VAR_GLOBAL

{attribute 'TcLinkTo' := 		'.q_xPress_OK		:= 	TIPC^txi_sxr_vac^txi_sxr_vac Instance^FSV_task Inputs^GVL_TXI_VAC_VFS.TV2K3_VFS_01.i_xPress_OK;
                                 .q_xOPN_SW			:=  TIPC^txi_sxr_vac^txi_sxr_vac Instance^FSV_task Inputs^GVL_TXI_VAC_VFS.TV2K3_VFS_01.i_xOPN_SW;
                                 .q_xCLS_SW			:=  TIPC^txi_sxr_vac^txi_sxr_vac Instance^FSV_task Inputs^GVL_TXI_VAC_VFS.TV2K3_VFS_01.i_xCLS_SW;
                                 .q_xVAC_FAULT_Reset:= 	TIPC^txi_sxr_vac^txi_sxr_vac Instance^FSV_task Inputs^GVL_TXI_VAC_VFS.TV2K3_VFS_01.i_xVAC_FAULT_Reset;
                                 .q_xOverrideMode	:= 	TIPC^txi_sxr_vac^txi_sxr_vac Instance^FSV_task Inputs^GVL_TXI_VAC_VFS.TV2K3_VFS_01.i_xOverrideMode;
                                 .q_xOverrideOpen	:= 	TIPC^txi_sxr_vac^txi_sxr_vac Instance^FSV_task Inputs^GVL_TXI_VAC_VFS.TV2K3_VFS_01.i_xOverrideOpen;
                                 .i_xTrigger		:=	TIPC^txi_sxr_vac^txi_sxr_vac Instance^FSV_task Outputs^GVL_TXI_VAC_VFS.TV2K3_VFS_01.q_xTrigger;
                                 .i_xVFS_Open		:=	TIPC^txi_sxr_vac^txi_sxr_vac Instance^FSV_task Outputs^GVL_TXI_VAC_VFS.TV2K3_VFS_01.q_xVFS_Open;
                                 .i_xVFS_Closed		:=	TIPC^txi_sxr_vac^txi_sxr_vac Instance^FSV_task Outputs^GVL_TXI_VAC_VFS.TV2K3_VFS_01.q_xVFS_Closed;
                                 .i_xVAC_FAULT_OK	:=  TIPC^txi_sxr_vac^txi_sxr_vac Instance^FSV_task Outputs^GVL_TXI_VAC_VFS.TV2K3_VFS_01.q_xVAC_FAULT_OK;
                                 .i_xMPS_OK			:=  TIPC^txi_sxr_vac^txi_sxr_vac Instance^FSV_task Outputs^GVL_TXI_VAC_VFS.TV2K3_VFS_01.q_xMPS_OK;
                                 .i_eVFS_State		:=	TIPC^txi_sxr_vac^txi_sxr_vac Instance^FSV_task Outputs^GVL_TXI_VAC_VFS.TV2K3_VFS_01.q_eVFS_State;
'}
TV2K3_VFS_01_Interface : FB_VFS_Interface;

{attribute 'pytmc' := 'pv: TV2K3:VFS:01'}
{attribute 'TcLinkTo' := 	'
        .q_xClose_A	:=	TIIB[H1K3S01-DRL-01 E1 (EL2202)]^Channel 1^Output;
        .q_xClose_B	:=	TIIB[H1K3S01-DRL-01 E1 (EL2202)]^Channel 2^Output;
        .q_xClose_C	:=	TIIB[H1K3S01-DRL-01 E2 (EL2202)]^Channel 1^Output;
        .q_xOPN_DO	:=	TIIB[H1K3S01-DRL-01 E2 (EL2202)]^Channel 2^Output;
        .i_xClsLS	:=	TIIB[H1K3S01-DRL-01 E3 (EL1004)]^Channel 1^Input;
        .i_xOpnLS	:=	TIIB[H1K3S01-DRL-01 E3 (EL1004)]^Channel 2^Input;
        .i_xTrigger :=  TIIB[E6 (EL1124)]^Channel 1^Input;
        .i_xPress_OK			:= 	TIPC^txi_sxr_vac^txi_sxr_vac Instance^PlcTask Outputs^GVL_TXI_VAC_VFS.TV2K3_VFS_01_Interface.q_xPRESS_OK;
        .i_xOPN_SW				:=  TIPC^txi_sxr_vac^txi_sxr_vac Instance^PlcTask Outputs^GVL_TXI_VAC_VFS.TV2K3_VFS_01_Interface.q_xOPN_SW;
        .i_xCLS_SW				:=  TIPC^txi_sxr_vac^txi_sxr_vac Instance^PlcTask Outputs^GVL_TXI_VAC_VFS.TV2K3_VFS_01_Interface.q_xCLS_SW;
        .i_xVAC_FAULT_Reset		:= 	TIPC^txi_sxr_vac^txi_sxr_vac Instance^PlcTask Outputs^GVL_TXI_VAC_VFS.TV2K3_VFS_01_Interface.q_xVAC_FAULT_Reset;
        .i_xOverrideMode		:= 	TIPC^txi_sxr_vac^txi_sxr_vac Instance^PlcTask Outputs^GVL_TXI_VAC_VFS.TV2K3_VFS_01_Interface.q_xOverrideMode;
        .i_xOverrideOpen		:= 	TIPC^txi_sxr_vac^txi_sxr_vac Instance^PlcTask Outputs^GVL_TXI_VAC_VFS.TV2K3_VFS_01_Interface.q_xOverrideOpen;
        .q_xTrigger				:=	TIPC^txi_sxr_vac^txi_sxr_vac Instance^PlcTask Inputs^GVL_TXI_VAC_VFS.TV2K3_VFS_01_Interface.i_xTrigger;
        .q_xVFS_Open			:=	TIPC^txi_sxr_vac^txi_sxr_vac Instance^PlcTask Inputs^GVL_TXI_VAC_VFS.TV2K3_VFS_01_Interface.i_xVFS_Open;
        .q_xVFS_Closed			:=	TIPC^txi_sxr_vac^txi_sxr_vac Instance^PlcTask Inputs^GVL_TXI_VAC_VFS.TV2K3_VFS_01_Interface.i_xVFS_Closed;
        .q_xVAC_FAULT_OK		:= 	TIPC^txi_sxr_vac^txi_sxr_vac Instance^PlcTask Inputs^GVL_TXI_VAC_VFS.TV2K3_VFS_01_Interface.i_xVAC_FAULT_OK;
        .q_xMPS_OK				:=  TIPC^txi_sxr_vac^txi_sxr_vac Instance^PlcTask Inputs^GVL_TXI_VAC_VFS.TV2K3_VFS_01_Interface.i_xMPS_OK;
        .q_eVFS_State			:=	TIPC^txi_sxr_vac^txi_sxr_vac Instance^PlcTask Inputs^GVL_TXI_VAC_VFS.TV2K3_VFS_01_Interface.i_eVFS_State;
        .i_xVetoValveOpenDO 	:= ;
        .i_xVetoValveClosed 	:=
'}
TV2K3_VFS_01 : FB_VFS;

END_VAR

(* stored: Version 1.1.0.1
   GVL GVL_TXI_VAC_VFS: Id {b5e2500d-8c0a-4623-a4a8-c639a1c0aee2} *)
